(* PLC project CoDeSys External Library Template, WAGO e!COCKPIT e!COCKPIT, author 3S - Smart Software Solutions GmbH *)
(* stored: creationDateTime 2019-10-29T12:37:19.4965558, version 3.5.5.30, modificationDateTime 2019-10-29T12:36:39.3744516, organization 3S - Smart Software Solutions GmbH *)
(* Library project template with all possible element types, docu and a sample project structure *)

{attribute 'qualified_only'}
{attribute 'strict'}
TYPE enumSystemError : (BrakHeartbetuzIZE := 1, NiezgodnaIloscKomunikatowOdebranychZIZE := 2, BladCRCWKomunikacieZIZE := 3, BladSzyfrowania := 4, ZaDuzaIloscKomunikatowWBuforze := 5, BladWalidacjiFullIdentifier := 6, BladFullIdentifierWHeartBeat := 7, BlokadaWysylaniaRamek := 8);
END_TYPE
